// TIA Portal project "Trapano" (V16)

(* hardware
DEVICE "S7-1200 station_1"  S7-1200 Station
   slot 0: "Telaio di montaggio_0"  S7-1200 Rack  Rack  V1.0
   slot 1: "PLC_1"  CPU 1214C DC/DC/DC  6ES7 214-1AG40-0XB0  V4.1
*)

// ===== PLC "PLC_1"  CPU 1214C DC/DC/DC =====

VAR_GLOBAL   // PLC tag table "Tabella delle variabili standard"
   "START" AT %I0.0 : Bool;
   "A" AT %I0.1 : Bool;
   "B" AT %I0.2 : Bool;
   "M" AT %I0.3 : Bool;
   "X" AT %I0.4 : Bool;
   "Y" AT %I0.5 : Bool;
   "DOWN" AT %Q0.0 : Bool;
   "UP" AT %Q0.1 : Bool;
   "RATATE" AT %Q0.2 : Bool;
   "OIL" AT %Q0.3 : Bool;
END_VAR

VAR_GLOBAL CONSTANT   // PLC tag table "Tabella delle variabili standard"
   "TEMPO_TRASCORSO" : Time := T#5s;
END_VAR

DATA_BLOCK "VariabiliDiStato"   // DB1
{ S7_Optimized_Access := 'TRUE' }
VERSION : 0.1
   VAR RETAIN
      HOME : Bool := true;
      SCENDI : Bool;
      Pezzo_Alto : Bool;
      Pezzo_Alto_Risalita : Bool;
      LUBRIFICA : Bool;
      FORO : Bool;
      SALI : Bool;
      WAIT : Bool;
   END_VAR
BEGIN
END_DATA_BLOCK

// folder: System blocks/Program resources

DATA_BLOCK "IEC_Timer_0_DB"   // DB2
{ S7_Optimized_Access := 'TRUE' }
AUTHOR : Simatic
FAMILY : IEC
NAME : IEC_TMR
VERSION : 1.0
// stored: InstanceOfName IEC_TIMER
"IEC_TIMER"
BEGIN
END_DATA_BLOCK

// folder: (top level)

ORGANIZATION_BLOCK "Main"   // OB1, LAD, ProgramCycle
TITLE = "Main Program Sweep (Cycle)"
{ S7_Optimized_Access := 'TRUE' }
VERSION : 0.1
   VAR_INPUT
      Initial_Call : Bool;   // Initial call of this OB
      Remanence : Bool;   // =True, if remanent data are available
   END_VAR
   VAR_TEMP   // added for the SCL form of the ladder/FBD networks
      _w1 : Bool;
   END_VAR
BEGIN

REGION Network 1
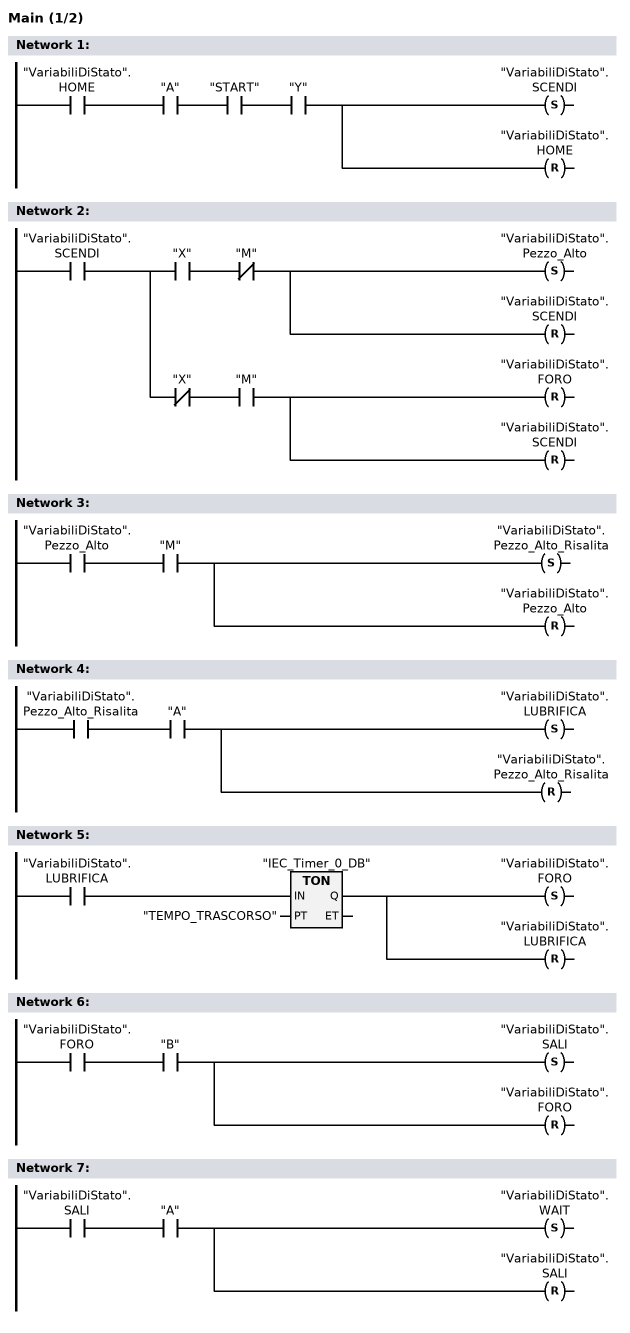
   RUNG wire#powerrail
      Contact( "VariabiliDiStato".HOME )
      Contact( "A" )
      Contact( "START" )
      Contact( "Y" )
      wire#w1
      S_Coil( "VariabiliDiStato".SCENDI )
   END_RUNG
   RUNG wire#w1
      R_Coil( "VariabiliDiStato".HOME )
   END_RUNG
   // the same network as SCL:
   IF "VariabiliDiStato".HOME AND "A" AND "START" AND "Y" THEN
       "VariabiliDiStato".SCENDI := TRUE;
       "VariabiliDiStato".HOME := FALSE;
   END_IF;
END_REGION

REGION Network 2
   RUNG wire#powerrail
      Contact( "VariabiliDiStato".SCENDI )
      wire#w1
      Contact( "X" )
      I_Contact( "M" )
      wire#w2
      S_Coil( "VariabiliDiStato".Pezzo_Alto )
   END_RUNG
   RUNG wire#w2
      R_Coil( "VariabiliDiStato".SCENDI )
   END_RUNG
   RUNG wire#w1
      I_Contact( "X" )
      Contact( "M" )
      wire#w3
      R_Coil( "VariabiliDiStato".FORO )
   END_RUNG
   RUNG wire#w3
      R_Coil( "VariabiliDiStato".SCENDI )
   END_RUNG
   // the same network as SCL:
   IF "VariabiliDiStato".SCENDI AND "X" AND NOT "M" THEN "VariabiliDiStato".Pezzo_Alto := TRUE; END_IF;
   #_w1 := "VariabiliDiStato".SCENDI;
   IF "VariabiliDiStato".SCENDI AND "X" AND NOT "M" THEN "VariabiliDiStato".SCENDI := FALSE; END_IF;
   IF #_w1 AND NOT "X" AND "M" THEN
       "VariabiliDiStato".FORO := FALSE;
       "VariabiliDiStato".SCENDI := FALSE;
   END_IF;
END_REGION

REGION Network 3
   RUNG wire#powerrail
      Contact( "VariabiliDiStato".Pezzo_Alto )
      Contact( "M" )
      wire#w1
      S_Coil( "VariabiliDiStato".Pezzo_Alto_Risalita )
   END_RUNG
   RUNG wire#w1
      R_Coil( "VariabiliDiStato".Pezzo_Alto )
   END_RUNG
   // the same network as SCL:
   IF "VariabiliDiStato".Pezzo_Alto AND "M" THEN
       "VariabiliDiStato".Pezzo_Alto_Risalita := TRUE;
       "VariabiliDiStato".Pezzo_Alto := FALSE;
   END_IF;
END_REGION

REGION Network 4
   RUNG wire#powerrail
      Contact( "VariabiliDiStato".Pezzo_Alto_Risalita )
      Contact( "A" )
      wire#w1
      S_Coil( "VariabiliDiStato".LUBRIFICA )
   END_RUNG
   RUNG wire#w1
      R_Coil( "VariabiliDiStato".Pezzo_Alto_Risalita )
   END_RUNG
   // the same network as SCL:
   IF "VariabiliDiStato".Pezzo_Alto_Risalita AND "A" THEN
       "VariabiliDiStato".LUBRIFICA := TRUE;
       "VariabiliDiStato".Pezzo_Alto_Risalita := FALSE;
   END_IF;
END_REGION

REGION Network 5
   "IEC_Timer_0_DB".TON(IN := "VariabiliDiStato".LUBRIFICA, PT := "TEMPO_TRASCORSO");
   IF "IEC_Timer_0_DB".Q THEN
       "VariabiliDiStato".FORO := TRUE;
       "VariabiliDiStato".LUBRIFICA := FALSE;
   END_IF;
END_REGION

REGION Network 6
   RUNG wire#powerrail
      Contact( "VariabiliDiStato".FORO )
      Contact( "B" )
      wire#w1
      S_Coil( "VariabiliDiStato".SALI )
   END_RUNG
   RUNG wire#w1
      R_Coil( "VariabiliDiStato".FORO )
   END_RUNG
   // the same network as SCL:
   IF "VariabiliDiStato".FORO AND "B" THEN
       "VariabiliDiStato".SALI := TRUE;
       "VariabiliDiStato".FORO := FALSE;
   END_IF;
END_REGION

REGION Network 7
   RUNG wire#powerrail
      Contact( "VariabiliDiStato".SALI )
      Contact( "A" )
      wire#w1
      S_Coil( "VariabiliDiStato".WAIT )
   END_RUNG
   RUNG wire#w1
      R_Coil( "VariabiliDiStato".SALI )
   END_RUNG
   // the same network as SCL:
   IF "VariabiliDiStato".SALI AND "A" THEN
       "VariabiliDiStato".WAIT := TRUE;
       "VariabiliDiStato".SALI := FALSE;
   END_IF;
END_REGION

REGION Network 8
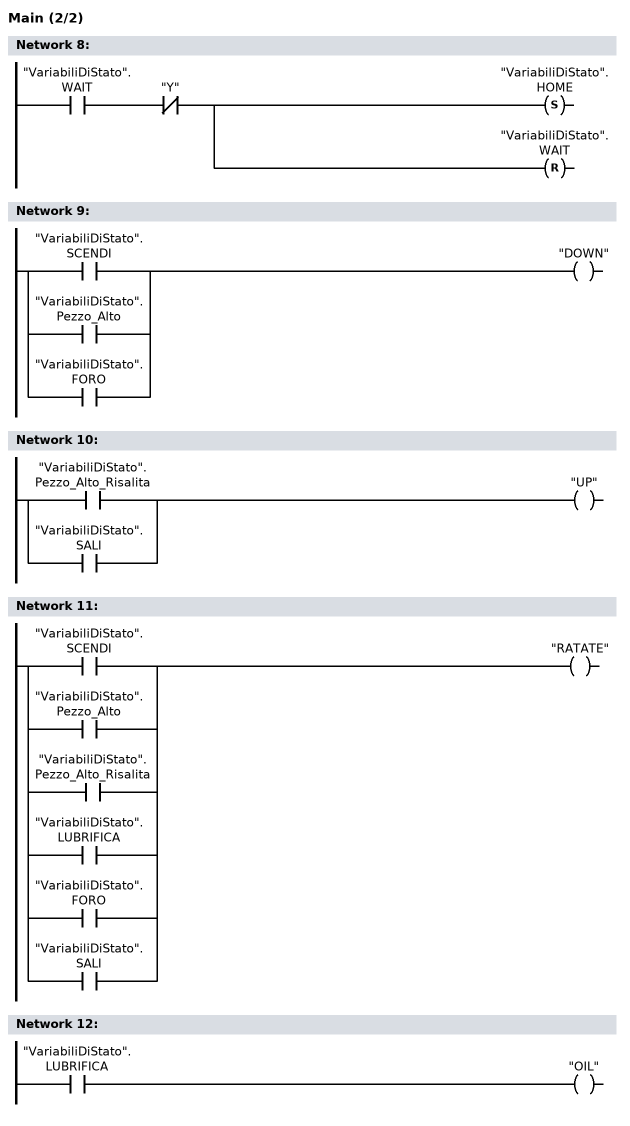
   RUNG wire#powerrail
      Contact( "VariabiliDiStato".WAIT )
      I_Contact( "Y" )
      wire#w1
      S_Coil( "VariabiliDiStato".HOME )
   END_RUNG
   RUNG wire#w1
      R_Coil( "VariabiliDiStato".WAIT )
   END_RUNG
   // the same network as SCL:
   IF "VariabiliDiStato".WAIT AND NOT "Y" THEN
       "VariabiliDiStato".HOME := TRUE;
       "VariabiliDiStato".WAIT := FALSE;
   END_IF;
END_REGION

REGION Network 9
   RUNG wire#powerrail
      Contact( "VariabiliDiStato".SCENDI )
      wire#w1
      Coil( "DOWN" )
   END_RUNG
   RUNG wire#powerrail
      Contact( "VariabiliDiStato".Pezzo_Alto )
   END_RUNG wire#w1
   RUNG wire#powerrail
      Contact( "VariabiliDiStato".FORO )
   END_RUNG wire#w1
   // the same network as SCL:
   "DOWN" := "VariabiliDiStato".SCENDI OR "VariabiliDiStato".Pezzo_Alto OR "VariabiliDiStato".FORO;
END_REGION

REGION Network 10
   RUNG wire#powerrail
      Contact( "VariabiliDiStato".Pezzo_Alto_Risalita )
      wire#w1
      Coil( "UP" )
   END_RUNG
   RUNG wire#powerrail
      Contact( "VariabiliDiStato".SALI )
   END_RUNG wire#w1
   // the same network as SCL:
   "UP" := "VariabiliDiStato".Pezzo_Alto_Risalita OR "VariabiliDiStato".SALI;
END_REGION

REGION Network 11
   RUNG wire#powerrail
      Contact( "VariabiliDiStato".SCENDI )
      wire#w1
      Coil( "RATATE" )
   END_RUNG
   RUNG wire#powerrail
      Contact( "VariabiliDiStato".Pezzo_Alto )
   END_RUNG wire#w1
   RUNG wire#powerrail
      Contact( "VariabiliDiStato".Pezzo_Alto_Risalita )
   END_RUNG wire#w1
   RUNG wire#powerrail
      Contact( "VariabiliDiStato".LUBRIFICA )
   END_RUNG wire#w1
   RUNG wire#powerrail
      Contact( "VariabiliDiStato".FORO )
   END_RUNG wire#w1
   RUNG wire#powerrail
      Contact( "VariabiliDiStato".SALI )
   END_RUNG wire#w1
   // the same network as SCL:
   "RATATE" := "VariabiliDiStato".SCENDI OR "VariabiliDiStato".Pezzo_Alto OR "VariabiliDiStato".Pezzo_Alto_Risalita OR "VariabiliDiStato".LUBRIFICA OR "VariabiliDiStato".FORO OR "VariabiliDiStato".SALI;
END_REGION

REGION Network 12
   RUNG wire#powerrail
      Contact( "VariabiliDiStato".LUBRIFICA )
      Coil( "OIL" )
   END_RUNG
   // the same network as SCL:
   "OIL" := "VariabiliDiStato".LUBRIFICA;
END_REGION
END_ORGANIZATION_BLOCK